PROGRAM p10_ladder
VAR
	bServoLadder: BOOL;
END_VAR

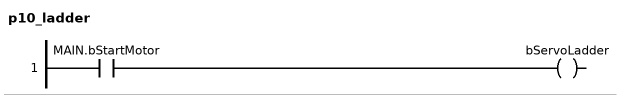
// NETWORK 1
bServoLadder := MAIN.bStartMotor;

END_PROGRAM

(* stored: Version 1.1.0.1, ProductVersion 3.1.4024.13
   POU p10_ladder: Id {37ff910e-7019-47b9-987e-eafc24eaf396}, SpecialFunc None *)
